// TIA Portal V17 export
// export: Created 2023-12-22T15:08:09.9188303Z, ExportSetting WithDefaults, DisplayName Totally Integrated Automation Portal, DisplayVersion V17, DisplayName TIA Portal Openness, DisplayVersion V17, DisplayName TIA Portal Version Control Interface, DisplayVersion V17, DisplayName STEP 7 Professional, DisplayVersion V17, DisplayName STEP 7 Safety, DisplayVersion V17, DisplayName WinCC Advanced, DisplayVersion V17
DATA_BLOCK "Any_DB"   // DB50
{ S7_Optimized_Access := 'FALSE' }
VERSION : 0.1
// stored: AutoNumber false, DBAccessibleFromOPCUA true, DBAccessibleFromWebserver true, IsOnlyStoredInLoadMemory false, IsWriteProtectedInAS false
   VAR RETAIN
      LE_1 : Real;
      LE_2 : Real;
      LE_3 : Real;
      LE_4 : Real;
      SP_TE_1 { S7_SetPoint := 'True'} : Real := 22.0;
      SP_TE_2 { S7_SetPoint := 'True'} : Real := 22.0;
      PS_Cl_1 : Bool;
      PS_Cl_2 : Bool;
   END_VAR
BEGIN
END_DATA_BLOCK
